FUNCTION_BLOCK TestADSLogger EXTENDS TcUnit.FB_TestSuite
VAR_INPUT
END_VAR
VAR_OUTPUT
END_VAR
VAR
END_VAR

submit_info();
submit_warning();
submit_error();
submit_alarm();

METHOD submit_alarm
VAR_INPUT
END_VAR
VAR_INST
  sut: ADSLoggerTestsystem;
END_VAR
TEST('Submit alarm');

sut.runner.add_logger(sut.logger);
sut.event.message := 'Alarm';
sut.event.alarm();

TEST_FINISHED();
END_METHOD

METHOD submit_error
VAR_INPUT
END_VAR
VAR_INST
  sut: ADSLoggerTestsystem;
END_VAR
TEST('Submit error');

sut.runner.add_logger(sut.logger);
sut.event.message := 'Error';
sut.event.error();

TEST_FINISHED();
END_METHOD

METHOD submit_info
VAR_INPUT
END_VAR
VAR_INST
  sut: ADSLoggerTestsystem;
END_VAR
TEST('Submit info');

sut.runner.add_logger(sut.logger);
sut.event.message := 'Info';
sut.event.info();

TEST_FINISHED();
END_METHOD

METHOD submit_warning
VAR_INPUT
END_VAR
VAR_INST
  sut: ADSLoggerTestsystem;
END_VAR
TEST('Submit warning');

sut.runner.add_logger(sut.logger);
sut.event.message := 'Warning';
sut.event.warning();

TEST_FINISHED();
END_METHOD

END_FUNCTION_BLOCK

(* stored: Version 1.1.0.1, ProductVersion 3.1.4024.9
   POU TestADSLogger: Id {e126a8bd-dc53-47fb-b987-2c50fb609a8b}, SpecialFunc None
   Method submit_alarm: Id {7203e8ee-f5fe-4e56-af12-ce30cf3bab16}
   Method submit_error: Id {7c89dd55-cac3-43cf-b229-89629492e809}
   Method submit_info: Id {bd81e84a-3e0d-47ff-97fa-d790029e78ab}
   Method submit_warning: Id {d791f11d-b6d0-4afa-8f91-e5b068e59d16} *)
